Fanuc KAREL source: kt00599.KL

-- PROVISIONAL review KL for V1013-1; original PC SHA256 40a6eb82388ce54f8752bc6eb554fdcbc7c1b86662d001027beb5092aca811c6
-- Incomplete behavior may be omitted. Consult companion uncertainty JSON. Do not deploy.
PROGRAM KT00599
%NOLOCKGROUP
VAR
  I1 : INTEGER
  I2 : INTEGER
  OUT : REAL
BEGIN
  -- UNRESOLVED_PC offsets 5-16; opcodes 2E,23
  -- UNRESOLVED_PC offsets 21-32; opcodes 2E,23
  -- UNRESOLVED_PC offsets 37-48; opcodes 2E,23
  -- UNRESOLVED_PC offsets 53-64; opcodes 2E,23
  -- UNRESOLVED_PC offsets 69-83; opcodes 21,48,64,23
  -- UNRESOLVED_PC offsets 88-92; opcodes 7F
END KT00599
